PROGRAM MAIN
VAR
END_VAR

END_PROGRAM

(* stored: Version 1.1.0.1
   POU MAIN: Id {94414385-07de-44df-a055-e296174cc4f5} *)
